(* IEC 61131-3 sources: LabBench/POU/01_Inputs/FB, 4 files *)

(* ---- FB_FloatLevelSensorGroup.st ---- *)
(*==============================================================================
    Название:    FB_FloatLevelSensorGroup
    Автор:       Редько А.
    Дата:        2025-04-26
    Версия:      1.1

    Описание:    Функциональный блок для группы поплавковых датчиков уровня.
                 Группа состоит из трех датчиков, расположенных на различных
                 уровнях в емкости высотой 500 мм:
                 - Нижний: 150 мм
                 - Средний: 250 мм
                 - Верхний: 350 мм

                 Блок обрабатывает сигналы с датчиков, определяет текущий
                 уровень жидкости и проверяет корректность показаний.

                 Реализован как level-controlled (LCon) блок
==============================================================================*)
FUNCTION_BLOCK FB_FloatLevelSensorGroup (* LCon *)
VAR_INPUT
    bEnable: BOOL := TRUE;      (* Разрешение работы *)
    bLowLevelSensor: BOOL;      (* Сигнал с нижнего датчика (150 мм) *)
    bMidLevelSensor: BOOL;      (* Сигнал со среднего датчика (250 мм) *)
    bHighLevelSensor: BOOL;     (* Сигнал с верхнего датчика (350 мм) *)
    rTankHeightMM: REAL := 500.0; (* Высота емкости, мм *)
    bReset: BOOL;               (* Сброс ошибок *)
END_VAR
VAR_OUTPUT
    bValid: BOOL;               (* Данные достоверны *)
    bError: BOOL;               (* Флаг ошибки *)
    wErrorID: WORD;             (* Код ошибки *)
    bLowLevelActive: BOOL;      (* Активен нижний датчик (150 мм) *)
    bMidLevelActive: BOOL;      (* Активен средний датчик (250 мм) *)
    bHighLevelActive: BOOL;     (* Активен верхний датчик (350 мм) *)
    eStatus: E_Inputs_Status;   (* Статус датчика *)
    rLevelEstimationMM: REAL;   (* Оценка текущего уровня в мм *)
    rLevelPercent: REAL;        (* Оценка уровня в процентах от максимального *)
END_VAR
VAR
    (* Параметры датчиков *)
    rLowLevelHeightMM: REAL := 150.0;  (* Высота нижнего датчика, мм *)
    rMidLevelHeightMM: REAL := 250.0;  (* Высота среднего датчика, мм *)
    rHighLevelHeightMM: REAL := 350.0; (* Высота верхнего датчика, мм *)

    (* Внутренние переменные *)
    bSensorSequenceValid: BOOL;        (* Флаг валидности последовательности *)
    stDataInternal: ST_FloatLevelGroup_Data; (* Внутренняя структура данных для обратной совместимости *)
END_VAR
VAR CONSTANT
    (* Битовая маска для кодов ошибок *)
    ERR_NONE: WORD := 16#0000;              (* Нет ошибок *)
    ERR_CONFIG: WORD := 16#0001;            (* Ошибка конфигурации *)
    ERR_INVALID_SEQUENCE: WORD := 16#0002;  (* Нарушена последовательность срабатывания *)
END_VAR

(* ======================================================================== *)
(* Основная логика функционального блока                                    *)
(* ======================================================================== *)

(* Инициализация *)
bLowLevelActive := FALSE;
bMidLevelActive := FALSE;
bHighLevelActive := FALSE;
wErrorID := ERR_NONE;
bValid := FALSE;
bError := FALSE;

(* Проверка конфигурации *)
IF rTankHeightMM <= 0.0 THEN
    (* Некорректно задана высота емкости *)
    eStatus := STATUS_CONFIG_ERROR;
    wErrorID := wErrorID OR ERR_CONFIG;
    bError := TRUE;

ELSIF rLowLevelHeightMM <= 0.0 OR rMidLevelHeightMM <= 0.0 OR rHighLevelHeightMM <= 0.0 THEN
    (* Некорректно заданы высоты датчиков *)
    eStatus := STATUS_CONFIG_ERROR;
    wErrorID := wErrorID OR ERR_CONFIG;
    bError := TRUE;

ELSIF rLowLevelHeightMM >= rMidLevelHeightMM OR rMidLevelHeightMM >= rHighLevelHeightMM THEN
    (* Нарушена последовательность высот датчиков *)
    eStatus := STATUS_CONFIG_ERROR;
    wErrorID := wErrorID OR ERR_CONFIG;
    bError := TRUE;

ELSIF rHighLevelHeightMM >= rTankHeightMM THEN
    (* Верхний датчик выше высоты емкости *)
    eStatus := STATUS_CONFIG_ERROR;
    wErrorID := wErrorID OR ERR_CONFIG;
    bError := TRUE;

ELSIF NOT bEnable THEN
    (* Блок отключен - возвращаем нулевые значения *)
    eStatus := STATUS_OK;
    rLevelEstimationMM := 0.0;
    rLevelPercent := 0.0;
    wErrorID := ERR_NONE;
    bValid := FALSE;
    bError := FALSE;

ELSE
    (* Нормальная работа - обработка сигналов датчиков *)

    (* Копируем состояния датчиков *)
    bLowLevelActive := bLowLevelSensor;
    bMidLevelActive := bMidLevelSensor;
    bHighLevelActive := bHighLevelSensor;

    (* Проверка последовательности срабатывания датчиков *)
    (* Если верхний датчик активен, средний и нижний тоже должны быть активны *)
    (* Если средний датчик активен, нижний тоже должен быть активен *)
    bSensorSequenceValid := TRUE;

    IF bHighLevelActive AND (NOT bMidLevelActive OR NOT bLowLevelActive) THEN
        (* Верхний датчик активен, но средний или нижний - нет *)
        bSensorSequenceValid := FALSE;
    ELSIF bMidLevelActive AND NOT bLowLevelActive THEN
        (* Средний датчик активен, но нижний - нет *)
        bSensorSequenceValid := FALSE;
    END_IF;

    IF NOT bSensorSequenceValid THEN
        (* Нарушена последовательность срабатывания датчиков *)
        eStatus := STATUS_INVALID_SEQUENCE;
        wErrorID := wErrorID OR ERR_INVALID_SEQUENCE;
        bValid := FALSE;
        bError := TRUE;
    ELSE
        (* Последовательность корректна - определяем уровень *)
        bValid := TRUE;
        bError := FALSE;

        (* Устанавливаем базовый статус *)
        eStatus := STATUS_OK;

        (* Оценка уровня на основе активных датчиков *)
        IF bHighLevelActive THEN
            (* Все три датчика активны - высокий уровень *)
            rLevelEstimationMM := rHighLevelHeightMM;
        ELSIF bMidLevelActive THEN
            (* Активны нижний и средний датчики - средний уровень *)
            rLevelEstimationMM := rMidLevelHeightMM;
        ELSIF bLowLevelActive THEN
            (* Активен только нижний датчик - низкий уровень *)
            rLevelEstimationMM := rLowLevelHeightMM;
        ELSE
            (* Ни один датчик не активен - уровень ниже нижнего датчика *)
            rLevelEstimationMM := rLowLevelHeightMM / 2.0; (* Примерная оценка - половина высоты нижнего датчика *)
        END_IF;

        (* Расчет процентного значения от максимальной высоты *)
        IF rTankHeightMM > 0.0 THEN
            rLevelPercent := (rLevelEstimationMM / rTankHeightMM) * 100.0;
        ELSE
            rLevelPercent := 0.0;
        END_IF;
    END_IF;
END_IF;

(* Сброс ошибок по внешнему сигналу *)
IF bReset THEN
    eStatus := STATUS_OK;
    wErrorID := ERR_NONE;
    bValid := TRUE;
    bError := FALSE;
END_IF;

(* Для обратной совместимости заполняем структуру stDataInternal *)
stDataInternal.bLowLevelActive := bLowLevelActive;
stDataInternal.bMidLevelActive := bMidLevelActive;
stDataInternal.bHighLevelActive := bHighLevelActive;
stDataInternal.eStatus := eStatus;
stDataInternal.rLevelEstimationMM := rLevelEstimationMM;
stDataInternal.rLevelPercent := rLevelPercent;
stDataInternal.wErrorCode := wErrorID;
stDataInternal.bValid := bValid;

(* ---- FB_FlowSensor.st ---- *)
(*==============================================================================
    Название:    FB_FlowSensor
    Автор:       Редько А.
    Дата:        2025-04-27
    Версия:      1.1

    Описание:    Универсальный функциональный блок для расходомеров
                 с частотным/импульсным выходом.

                 Реализован как level-controlled (LCon) блок
==============================================================================*)
FUNCTION_BLOCK FB_FlowSensor (* LCon *)
VAR_INPUT
    bEnable: BOOL := TRUE;        (* Разрешение работы *)
    wPulseCounter: WORD;          (* Значение счетчика импульсов *)
    rPulsePerLiter: REAL;         (* Количество импульсов на литр *)
    tSampleTime: TIME := T#500MS; (* Время выборки для расчета расхода *)
    bReset: BOOL;                 (* Сброс счетчиков и ошибок *)
END_VAR
VAR_OUTPUT
    bValid: BOOL;                 (* Данные достоверны *)
    bError: BOOL;                 (* Флаг ошибки *)
    wErrorID: WORD;               (* Код ошибки *)
    rFlowLPM: REAL;               (* Расход в л/мин *)
    rFlowM3H: REAL;               (* Расход в м³/ч *)
    rTotalLiters: REAL;           (* Общий объем в литрах *)
    rFrequencyHz: REAL;           (* Частота импульсов в Гц *)
    eStatus: E_Inputs_Status;     (* Статус датчика *)
    dwPulseCount: DWORD;          (* Накопленное количество импульсов *)
    dwPulseDelta: DWORD;          (* Количество импульсов за период *)
END_VAR
VAR
    (* Переменные для обработки импульсов *)
    dwPrevPulseCount: DWORD;      (* Предыдущее значение счетчика импульсов *)
    dwCurrentPulseCount: DWORD;   (* Текущее значение счетчика импульсов *)
    dwTotalPulseCount: DWORD;     (* Общее количество импульсов с учетом переполнений *)
    dwOverflowCounter: DWORD;     (* Счетчик переполнений WORD *)

    bFirstCycle: BOOL := TRUE;    (* Флаг первого цикла *)

    tTimer: TON;                  (* Таймер для расчета расхода *)
    rSampleTimeInSec: REAL;       (* Время выборки в секундах *)

    (* Структура для обратной совместимости *)
    stDataInternal: ST_FlowSensor_Data;
END_VAR
VAR CONSTANT
    (* Битовая маска для кодов ошибок *)
    ERR_NONE: WORD := 16#0000;            (* Нет ошибок *)
    ERR_CONFIG: WORD := 16#0001;          (* Ошибка конфигурации *)
END_VAR

(* ======================================================================== *)
(* Основная логика функционального блока                                    *)
(* ======================================================================== *)

(* Инициализация *)
wErrorID := ERR_NONE;
bValid := FALSE;
bError := FALSE;

(* Проверка конфигурации *)
IF rPulsePerLiter <= 0.0 THEN
    (* Некорректно задан коэффициент пересчета *)
    eStatus := STATUS_CONFIG_ERROR;
    wErrorID := wErrorID OR ERR_CONFIG;
    bError := TRUE;

ELSIF NOT bEnable THEN
    (* Блок отключен - нулевые значения *)
    eStatus := STATUS_OK;
    rFlowLPM := 0.0;
    rFlowM3H := 0.0;
    rFrequencyHz := 0.0;
    wErrorID := ERR_NONE;
    bValid := FALSE;
    bError := FALSE;

ELSE
    (* Нормальная работа - обработка данных *)

    (* Преобразование WORD в DWORD *)
    dwCurrentPulseCount := WORD_TO_DWORD(wPulseCounter);

    (* Обработка первого вызова *)
    IF bFirstCycle THEN
        dwPrevPulseCount := dwCurrentPulseCount;
        dwTotalPulseCount := dwCurrentPulseCount;
        bFirstCycle := FALSE;
    END_IF;

    (* Обработка переполнения счетчика *)
    IF dwCurrentPulseCount < dwPrevPulseCount THEN
        (* Счетчик переполнился - добавляем 65536 (2^16) *)
        dwOverflowCounter := dwOverflowCounter + 65536;
    END_IF;

    (* Расчет общего количества импульсов *)
    dwTotalPulseCount := dwCurrentPulseCount + dwOverflowCounter;
    dwPulseCount := dwTotalPulseCount;

    (* Запуск таймера для расчета расхода *)
    tTimer(IN := TRUE, PT := tSampleTime);

    (* Расчет расхода по частоте импульсов *)
    IF tTimer.Q THEN
        (* Вычисление количества импульсов за период *)
        dwPulseDelta := dwTotalPulseCount - dwPrevPulseCount;
        dwPrevPulseCount := dwTotalPulseCount;

        (* Преобразование времени выборки в секунды *)
        rSampleTimeInSec := TIME_TO_REAL(tSampleTime) / 1000.0;

        (* Расчет частоты импульсов (Гц) *)
        rFrequencyHz := DWORD_TO_REAL(dwPulseDelta) / rSampleTimeInSec;

        (* Расчет расхода в л/мин - универсальная формула для любого расходомера *)
        rFlowLPM := (rFrequencyHz * 60.0) / rPulsePerLiter;

        (* Расчет расхода в м³/ч *)
        rFlowM3H := rFlowLPM * 0.06; (* 1 л/мин = 0.06 м³/ч *)

        (* Расчет общего объема в литрах (полезно для учебных целей) *)
        rTotalLiters := DWORD_TO_REAL(dwPulseCount) / rPulsePerLiter;

        (* Данные валидны *)
        bValid := TRUE;
        bError := FALSE;
        eStatus := STATUS_OK;

        (* Сброс таймера для следующего периода *)
        tTimer(IN := FALSE);
    END_IF;
END_IF;

(* Сброс по внешнему сигналу *)
IF bReset THEN
    dwPrevPulseCount := dwCurrentPulseCount;
    dwOverflowCounter := 0;
    rTotalLiters := 0.0;
    eStatus := STATUS_OK;
    wErrorID := ERR_NONE;
    bValid := TRUE;
    bError := FALSE;
END_IF;

(* Заполнение структуры для обратной совместимости *)
stDataInternal.rFlowLPM := rFlowLPM;
stDataInternal.rFlowM3H := rFlowM3H;
stDataInternal.rTotalLiters := rTotalLiters;
stDataInternal.rFrequencyHz := rFrequencyHz;
stDataInternal.eStatus := eStatus;
stDataInternal.wErrorCode := wErrorID;
stDataInternal.bValid := bValid;
stDataInternal.dwPulseCount := dwPulseCount;
stDataInternal.dwPulseDelta := dwPulseDelta;

(* ---- FB_HydroLevelSensor.st ---- *)
(*==============================================================================
    Название:    FB_HydroLevelSensor
    Автор:       Редько А.
    Дата:        2025-04-25
    Версия:      1.2

    Описание:    Функциональный блок для гидростатического
                 датчика уровня.

                 Входные сигналы получены после масштабирования в конфигурации ПЛК.
                 Блок пересчитывает давление в уровень жидкости (мм).

                 Реализован как level-controlled (LCon) блок
==============================================================================*)
FUNCTION_BLOCK FB_HydroLevelSensor (* LCon *)
VAR_INPUT
    bEnable: BOOL := TRUE;         (* Разрешение работы *)
    rPressurePa: REAL;             (* Давление от датчика после масштабирования, Па *)
    rMaxAllowedLevelMM: REAL;      (* Максимально допустимый уровень, мм *)
    rDensity: REAL := 1000.0;      (* Плотность жидкости, кг/м³ *)
    rGravity: REAL := 9.81;        (* Ускорение свободного падения, м/с² *)
    rLevelOffset: REAL := 0.0;     (* Смещение уровня, мм (если датчик ниже дна) *)
    bReset: BOOL;                  (* Сброс ошибок *)
END_VAR
VAR_OUTPUT
    bValid: BOOL;                  (* Данные достоверны *)
    bError: BOOL;                  (* Флаг ошибки *)
    wErrorID: WORD;                (* Код ошибки *)
    rLevelMM: REAL;                (* Уровень в мм *)
    rLevelPercent: REAL;           (* Уровень в процентах от максимального *)
    rRawPressurePa: REAL;          (* Исходное значение давления *)
    eStatus: E_Inputs_Status;      (* Статус датчика *)
END_VAR
VAR
    (* Системные переменные *)
    byStatus: BYTE;                (* Старший байт из переменной для анализа статуса *)
    rCalculatedLevelMM: REAL;      (* Вычисленный уровень до проверок *)

    (* Структура для обратной совместимости *)
    stDataInternal: ST_HydroLevel_Data;
END_VAR
VAR CONSTANT
    (* Константы для статусов аналогового входа (старший байт) *)
    ERR_NONE: BYTE := 16#00;           (* Ошибок нет *)
    ERR_INVALID: BYTE := 16#F1;        (* Результаты измерения заведомо неверны *)
    ERR_NOT_READY: BYTE := 16#F6;      (* Результаты измерения не готовы *)
    ERR_ABOVE_RANGE: BYTE := 16#FA;    (* Сигнал на входе больше возможного *)
    ERR_BELOW_RANGE: BYTE := 16#FB;    (* Сигнал на входе меньше возможного *)
    ERR_CURRENT_OVERLOAD: BYTE := 16#FC;(* Перегрузка в канале измерения тока *)
    ERR_VOLTAGE_BREAK: BYTE := 16#FD;  (* Обрыв датчика в канале измерения напряжения *)

    (* Битовая маска для кодов ошибок *)
    ERROR_CONFIG: WORD := 16#0001;           (* Ошибка конфигурации *)
    ERROR_VALUE_ABOVE_MAX: WORD := 16#0002;  (* Превышение макс. допустимого уровня *)
    ERROR_AI_ABOVE_RANGE: WORD := 16#0004;   (* Превышение диапазона аналогового входа *)
    ERROR_AI_BELOW_RANGE: WORD := 16#0008;   (* Значение ниже диапазона аналогового входа *)
    ERROR_WIRE_BREAK: WORD := 16#0010;       (* Обрыв линии датчика *)
    ERROR_CURRENT_OVERLOAD_MASK: WORD := 16#0020; (* Перегрузка в канале измерения тока *)
    ERROR_NOT_READY_MASK: WORD := 16#0040;   (* Измерение не готово *)
    ERROR_UNKNOWN: WORD := 16#8000;          (* Неизвестная ошибка *)
END_VAR

(* ======================================================================== *)
(* Основная логика функционального блока                                    *)
(* ======================================================================== *)

(* Инициализация *)
rRawPressurePa := rPressurePa;  (* Сохраняем исходное значение для диагностики *)
wErrorID := 0;
bValid := FALSE;
bError := FALSE;

(* Проверка конфигурации *)
IF rMaxAllowedLevelMM <= 0.0 THEN
    (* Некорректно задан максимальный допустимый уровень *)
    eStatus := STATUS_CONFIG_ERROR;
    wErrorID := wErrorID OR ERROR_CONFIG;
    bError := TRUE;

ELSIF rDensity <= 0.0 THEN
    (* Некорректно задана плотность жидкости *)
    eStatus := STATUS_CONFIG_ERROR;
    wErrorID := wErrorID OR ERROR_CONFIG;
    bError := TRUE;

ELSIF rGravity <= 0.0 THEN
    (* Некорректно задано ускорение свободного падения *)
    eStatus := STATUS_CONFIG_ERROR;
    wErrorID := wErrorID OR ERROR_CONFIG;
    bError := TRUE;

ELSIF NOT bEnable THEN
    (* Блок отключен - возвращаем нулевые значения *)
    eStatus := STATUS_OK;
    rLevelMM := 0.0;
    rLevelPercent := 0.0;
    wErrorID := 0;
    bValid := FALSE;
    bError := FALSE;

ELSE
    (* Нормальная работа - обработка данных и проверка ошибок *)

    (* Получение старшего байта для анализа статуса *)
    byStatus := DWORD_TO_BYTE(SHR(REAL_TO_DWORD(rPressurePa) AND 16#FF000000, 24));

    (* Проверка статуса аналогового входа *)
    CASE byStatus OF
        ERR_NONE:
            (* Нормальные данные - статус OK *)
            eStatus := STATUS_OK;
            bValid := TRUE;
            bError := FALSE;

        ERR_ABOVE_RANGE:
            (* Превышение диапазона аналогового входа *)
            eStatus := STATUS_AI_ABOVE_RANGE;
            wErrorID := wErrorID OR ERROR_AI_ABOVE_RANGE;
            bValid := FALSE;
            bError := TRUE;

        ERR_BELOW_RANGE:
            (* Значение ниже диапазона аналогового входа *)
            eStatus := STATUS_AI_BELOW_RANGE;
            wErrorID := wErrorID OR ERROR_AI_BELOW_RANGE;
            bValid := FALSE;
            bError := TRUE;

        ERR_VOLTAGE_BREAK:
            (* Обрыв линии датчика *)
            eStatus := STATUS_WIRE_BREAK;
            wErrorID := wErrorID OR ERROR_WIRE_BREAK;
            bValid := FALSE;
            bError := TRUE;

        ERR_CURRENT_OVERLOAD:
            (* Перегрузка в канале измерения тока *)
            eStatus := STATUS_CURRENT_OVERLOAD;
            wErrorID := wErrorID OR ERROR_CURRENT_OVERLOAD_MASK;
            bValid := FALSE;
            bError := TRUE;

        ERR_NOT_READY:
            (* Измерение не готово *)
            eStatus := STATUS_NOT_READY;
            wErrorID := wErrorID OR ERROR_NOT_READY_MASK;
            bValid := FALSE;
            bError := TRUE;

        ELSE
            (* Прочие неизвестные ошибки *)
            eStatus := STATUS_UNKNOWN;
            wErrorID := wErrorID OR ERROR_UNKNOWN;
            bValid := FALSE;
            bError := TRUE;
    END_CASE;

    (* Расчет уровня по гидростатической формуле: h = P / (ρ * g) *)
    (* Проверка деления на ноль *)
    IF rDensity * rGravity > 0.001 THEN
        (* Перевод метров в миллиметры (умножение на 1000) *)
        rCalculatedLevelMM := (rPressurePa / (rDensity * rGravity)) * 1000.0;

        (* Добавление смещения уровня (для коррекции положения датчика) *)
        rCalculatedLevelMM := rCalculatedLevelMM + rLevelOffset;

        (* Ограничение снизу нулем - уровень не может быть отрицательным *)
        rLevelMM := MAX(0.0, rCalculatedLevelMM);

        (* Расчет процентного значения от максимального уровня *)
        IF rMaxAllowedLevelMM > 0.0 THEN
            rLevelPercent := (rLevelMM / rMaxAllowedLevelMM) * 100.0;
        ELSE
            rLevelPercent := 0.0;
        END_IF;
    ELSE
        (* Ошибка деления на ноль из-за конфигурации *)
        rLevelMM := 0.0;
        rLevelPercent := 0.0;
        eStatus := STATUS_CONFIG_ERROR;
        wErrorID := wErrorID OR ERROR_CONFIG;
        bValid := FALSE;
        bError := TRUE;
    END_IF;

    (* Проверка на превышение максимально допустимого уровня емкости *)
    IF rLevelMM > rMaxAllowedLevelMM AND rMaxAllowedLevelMM > 0.0 THEN
        (* Выставляем ошибку превышения физического уровня *)
        eStatus := STATUS_VALUE_ABOVE_MAX;
        wErrorID := wErrorID OR ERROR_VALUE_ABOVE_MAX;
        bValid := FALSE;
        bError := TRUE;
    END_IF;
END_IF;

(* Сброс ошибок по внешнему сигналу *)
IF bReset THEN
    eStatus := STATUS_OK;
    wErrorID := 0;
    bValid := TRUE;
    bError := FALSE;
END_IF;

(* Заполнение структуры для обратной совместимости *)
stDataInternal.rLevelMM := rLevelMM;
stDataInternal.rLevelPercent := rLevelPercent;
stDataInternal.eStatus := eStatus;
stDataInternal.wErrorCode := wErrorID;
stDataInternal.bValid := bValid;
stDataInternal.rRawPressurePa := rRawPressurePa;

(* ---- FB_PressureSensor.st ---- *)
(*==============================================================================
    Название:    FB_PressureSensor
    Автор:       Редько А.
    Дата:        2025-04-25
    Версия:      1.2

    Описание:    Функциональный блок для датчиков давления.

                 Данные получаются после масштабирования в конфигурации ПЛК.
                 Блок проверяет статус измерения, выполняет проверку на
                 превышение предельного значения и формирует результаты.

                 Фильтрация и обработка статусов выполняется в конфигурации ПЛК

                 Реализован как level-controlled (LCon) блок
==============================================================================*)
FUNCTION_BLOCK FB_PressureSensor (* LCon *)
VAR_INPUT
    bEnable: BOOL := TRUE;      (* Разрешение работы *)
    rPressureKPa: REAL;         (* Давление в кПа (с аналогового входа после масштабирования) *)
    rMaxPressureKPa: REAL;      (* Максимально допустимое давление, кПа *)
    bReset: BOOL;               (* Сброс ошибок *)
END_VAR

VAR_OUTPUT
    bValid: BOOL;               (* Данные достоверны *)
    bError: BOOL;               (* Флаг ошибки *)
    wErrorID: WORD;             (* Код ошибки *)
    rPressureValue: REAL;       (* Давление в кПа *)
    eStatus: E_Inputs_Status;   (* Статус датчика *)
END_VAR

VAR
    (* Системные переменные *)
    byStatus: BYTE;             (* Старший байт из переменной для анализа статуса *)

    (* Структура для обратной совместимости *)
    stDataInternal: ST_PressureSensor_Data;
END_VAR

VAR CONSTANT
    (* Константы для статусов аналогового входа (старший байт) *)
    ERR_NONE: BYTE := 16#00;           (* Ошибок нет *)
    ERR_INVALID: BYTE := 16#F1;        (* Результаты измерения заведомо неверны *)
    ERR_NOT_READY: BYTE := 16#F6;      (* Результаты измерения не готовы *)
    ERR_ABOVE_RANGE: BYTE := 16#FA;    (* Сигнал на входе больше возможного *)
    ERR_BELOW_RANGE: BYTE := 16#FB;    (* Сигнал на входе меньше возможного *)
    ERR_CURRENT_OVERLOAD: BYTE := 16#FC;(* Перегрузка в канале измерения тока *)
    ERR_VOLTAGE_BREAK: BYTE := 16#FD;  (* Обрыв датчика в канале измерения напряжения *)

    (* Битовые маски для кодов ошибок *)
    ERROR_NONE: WORD := 16#0000;           (* Нет ошибок *)
    ERROR_CONFIG: WORD := 16#0001;         (* Ошибка конфигурации *)
    ERROR_VALUE_ABOVE_MAX: WORD := 16#0002;    (* Превышение максимального давления *)
    ERROR_AI_ABOVE_RANGE: WORD := 16#0004; (* Превышение диапазона аналогового входа *)
    ERROR_AI_BELOW_RANGE: WORD := 16#0008; (* Значение ниже диапазона аналогового входа *)
    ERROR_WIRE_BREAK: WORD := 16#0010;     (* Обрыв линии датчика *)
    ERROR_CURRENT_OVERLOAD: WORD := 16#0020; (* Перегрузка в канале измерения тока *)
    ERROR_NOT_READY: WORD := 16#0040;      (* Измерение не готово *)
    ERROR_UNKNOWN: WORD := 16#8000;        (* Неизвестная ошибка *)
END_VAR

(* ======================================================================== *)
(* Основная логика функционального блока                                    *)
(* ======================================================================== *)

(* Инициализация *)
rPressureValue := rPressureKPa;  (* Сохраняем исходное значение *)
wErrorID := ERROR_NONE;
bValid := FALSE;
bError := FALSE;

(* Проверка конфигурации *)
IF rMaxPressureKPa <= 0.0 THEN
    (* Некорректно задано максимальное давление *)
    eStatus := STATUS_CONFIG_ERROR;
    wErrorID := wErrorID OR ERROR_CONFIG;
    bError := TRUE;

ELSIF NOT bEnable THEN
    (* Блок отключен - возвращаем нулевые значения *)
    eStatus := STATUS_OK;
    rPressureValue := 0.0;
    wErrorID := ERROR_NONE;
    bValid := FALSE;
    bError := FALSE;

ELSE
    (* Нормальная работа - обработка данных и проверка ошибок *)

    (* Получение старшего байта для анализа статуса *)
    byStatus := DWORD_TO_BYTE(SHR(REAL_TO_DWORD(rPressureKPa) AND 16#FF000000, 24));

    (* Проверка статуса аналогового входа *)
    CASE byStatus OF
        ERR_NONE:
            (* Нормальные данные - статус OK *)
            eStatus := STATUS_OK;
            bValid := TRUE;
            bError := FALSE;

        ERR_ABOVE_RANGE:
            (* Превышение диапазона аналогового входа *)
            eStatus := STATUS_AI_ABOVE_RANGE;
            wErrorID := wErrorID OR ERROR_AI_ABOVE_RANGE;
            bValid := FALSE;
            bError := TRUE;

        ERR_BELOW_RANGE:
            (* Значение ниже диапазона аналогового входа *)
            eStatus := STATUS_AI_BELOW_RANGE;
            wErrorID := wErrorID OR ERROR_AI_BELOW_RANGE;
            bValid := FALSE;
            bError := TRUE;

        ERR_VOLTAGE_BREAK:
            (* Обрыв линии датчика *)
            eStatus := STATUS_WIRE_BREAK;
            wErrorID := wErrorID OR ERROR_WIRE_BREAK;
            bValid := FALSE;
            bError := TRUE;

        ERR_CURRENT_OVERLOAD:
            (* Перегрузка в канале измерения тока *)
            eStatus := STATUS_CURRENT_OVERLOAD;
            wErrorID := wErrorID OR ERROR_CURRENT_OVERLOAD;
            bValid := FALSE;
            bError := TRUE;

        ERR_NOT_READY:
            (* Измерение не готово *)
            eStatus := STATUS_NOT_READY;
            wErrorID := wErrorID OR ERROR_NOT_READY;
            bValid := FALSE;
            bError := TRUE;

        ELSE
            (* Прочие неизвестные ошибки *)
            eStatus := STATUS_UNKNOWN;
            wErrorID := wErrorID OR ERROR_UNKNOWN;
            bValid := FALSE;
            bError := TRUE;
    END_CASE;

    (* Проверка на превышение максимально допустимого давления *)
    IF rPressureKPa > rMaxPressureKPa AND rMaxPressureKPa > 0.0 AND bValid THEN
        (* Выставляем ошибку превышения давления *)
        eStatus := STATUS_VALUE_ABOVE_MAX;
        wErrorID := wErrorID OR ERROR_VALUE_ABOVE_MAX;
        bValid := FALSE;
        bError := TRUE;
    END_IF;
END_IF;

(* Сброс ошибок по внешнему сигналу *)
IF bReset THEN
    eStatus := STATUS_OK;
    wErrorID := ERROR_NONE;
    bValid := TRUE;
    bError := FALSE;
END_IF;

(* Заполнение структуры для обратной совместимости *)
stDataInternal.rPressureKPa := rPressureValue;
stDataInternal.eStatus := eStatus;
stDataInternal.wErrorCode := wErrorID;
stDataInternal.bValid := bValid;
